TYPE E_StepperState :
	
(
	Offline,
	Reset,
	Power,
	Error,
	Operational,
	EncHoming,
	Homing,
	Jog
);

END_TYPE

(* stored: Version 1.1.0.1
   DUT E_StepperState: Id {4de45bb8-fc09-4ba5-adbb-27018f9f93fc} *)
